FUNCTION_BLOCK FB_SodaFill IMPLEMENTS I_FillingStrategy
VAR_INPUT
END_VAR
VAR_OUTPUT
END_VAR
VAR
END_VAR

{warning 'add method implementation '}
METHOD ExecuteFill : BOOL
VAR_INPUT
	stBottle : REFERENCE TO ST_Bottle;
END_VAR

VAR CONSTANT
	cFILLING_SPEED: REAL:= 5;
END_VAR
IF __ISVALIDREF(stBottle) THEN
	IF stBottle.fCurrentLevel >= stBottle.fTargetLevel THEN
		ExecuteFill := TRUE;
	ELSE
		stBottle.fCurrentLevel := stBottle.fCurrentLevel + cFILLING_SPEED;
		ExecuteFill := FALSE;
	END_IF
END_IF
END_METHOD

END_FUNCTION_BLOCK

(* stored: Version 1.1.0.1, ProductVersion 3.1.4024.16
   POU FB_SodaFill: Id {e0355c25-9e08-4871-88cd-6d5a8519cbc8}, SpecialFunc None
   Method ExecuteFill: Id {8f8533fc-0f23-43e7-8222-204e4f12ea9e} *)
